Yaskawa INFORM job: OK_R2_O22-23(-90,180)OKKR.JBI

/JOB
//NAME OK_R2_O22-23(-90,180)OKKR
///FOLDERNAME X4
//POS
///NPOS 109,109,109,5,0,0
///TOOL 0
///POSTYPE PULSE
///PULSE
C00000=34467,8161,-3438,41001,63186,-12360
C00001=79400,-96450,-73119,47071,38510,-50576
C00002=120689,-37236,-43262,1430,36977,-65337
C00003=120661,8390,6118,1752,30038,-65509
C00004=121363,14227,14389,901,27936,-65072
C00005=121630,18134,20803,569,25994,-64899
C00006=122051,20456,22985,-52,25844,-64579
C00007=122335,22651,22887,209,31352,-64420
C00008=122335,23153,24532,213,30597,-64422
C00009=122573,22007,22272,-73,31399,-64269
C00010=118553,33336,34533,-32200,31167,-63632
C00011=118554,33797,35647,-32601,30785,-63423
C00012=118795,35881,37778,-33055,30674,-63177
C00013=119029,34698,36884,-33342,30719,-63021
C00014=119029,35470,39068,-34241,29924,-62556
C00015=119029,34698,36884,-33342,30719,-63021
C00016=122566,16275,19454,-818,25870,-64189
C00017=120682,5973,-10666,-26006,48512,-34380
C00018=120682,6077,-8041,-26626,47105,-33962
C00019=120965,19546,-3322,-22995,60520,-37308
C00020=120686,6056,-8291,-26571,47234,-33999
C00021=120521,4024,-8795,-26757,46523,-33864
C00022=122243,21545,4650,-37838,56763,-29509
C00023=115724,34900,14421,-35017,60862,-31707
C00024=115313,34877,14397,-34830,60697,-31836
C00025=122685,12952,-4874,-39297,55027,-28576
C00026=131885,-4518,-22891,-42927,60902,-26587
C00027=120689,-37236,-43262,1430,36977,-65337
C00028=79400,-96450,-73119,47071,38510,-50576
C00029=-8645,-72931,-67050,57733,95594,-74029
C00030=-3643,-76224,-106676,-19950,71810,-76872
C00031=-266,-73751,-67438,57600,90404,-72524
C00032=56065,-40103,-98025,15235,73272,-62938
C00033=80290,13979,-35130,8518,69424,-54762
C00034=81621,16186,-30024,7817,67316,-54480
C00035=82138,17140,-27919,7543,66474,-54366
C00036=82701,19213,-25983,7203,66302,-54190
C00037=82138,17140,-27919,7543,66474,-54366
C00038=82074,13923,-28800,7646,65378,-54460
C00039=82073,13446,-28104,7686,64710,-54504
C00040=82074,14344,-29367,7613,65938,-54423
C00041=80200,10192,-35655,8662,67827,-54907
C00042=80279,11679,-32768,3860,64531,-54120
C00043=80277,10318,-30958,3920,62722,-54182
C00044=80747,9882,-30077,3637,61936,-54046
C00045=80280,10347,-31011,3916,62769,-54180
C00046=79691,8209,-31623,4330,62077,-54408
C00047=80388,10283,-29809,3872,61992,-54168
C00048=75041,22104,-18783,7439,61626,-56057
C00049=80303,10454,-30913,3901,62763,-54172
C00050=80304,11819,-32719,3842,64572,-54110
C00051=56065,-40103,-98025,15235,73272,-62938
C00052=-3643,-76224,-106676,-19950,71810,-76872
C00053=-266,-73751,-67438,57600,90404,-72524
C00054=-266,-73751,-67438,57600,90404,-72524
C00055=-266,-73751,-67438,57600,90404,-72524
C00056=-266,-73751,-67438,57600,90404,-72524
C00057=-266,-73751,-67438,57600,90404,-72524
C00058=-266,-73751,-67438,57600,90404,-72524
C00059=-266,-73751,-67438,57600,90404,-72524
C00060=-266,-73751,-67438,57600,90404,-72524
C00061=-266,-73751,-67438,57600,90404,-72524
C00062=120677,-3480,-20614,18181,54095,39471
C00063=120311,11594,-4773,18885,52273,38972
C00064=120169,13967,1466,19666,49827,38417
C00065=119883,15460,2829,19877,49828,38285
C00066=119880,14569,2014,19868,49870,38293
C00067=119880,14692,3030,20029,49339,38180
C00068=119880,15002,5218,20385,48223,37938
C00069=119880,14692,3030,20029,49339,38180
C00070=121128,7117,-4698,18949,49860,38864
C00071=120984,8550,-10493,36755,60982,29079
C00072=120492,10444,-8592,38530,61785,27976
C00073=119910,12056,-7149,38807,61994,27785
C00074=120247,11117,-7991,38646,61874,27896
C00075=120247,11130,-6123,39024,60976,27528
C00076=120247,11117,-7991,38646,61874,27896
C00077=118757,6782,-7537,20091,51910,38210
C00078=120681,6612,-10378,25984,47448,35852
C00079=120681,6707,-7755,26629,46038,35426
C00080=120905,16102,-4997,22232,56693,38204
C00081=120839,4648,-8519,26766,45460,35327
C00082=120685,6692,-7997,26566,46163,35467
C00083=117786,13784,-6304,24852,56256,36873
C00084=124524,9883,-9298,30535,58908,31643
C00085=123624,18800,-2226,35492,64552,29693
C00086=120681,6624,-6675,42630,54896,24176
C00087=115739,6767,-11022,43739,59328,23743
C00088=-266,-73751,-67438,57600,90404,-72524
C00089=-266,-73751,-67438,57600,90404,-72524
C00090=73074,14271,-65905,40005,100084,34925
C00091=80386,15191,-35510,35923,83035,31364
C00092=81077,18148,-29671,35761,81084,30977
C00093=80079,11495,-28631,39585,73800,28709
C00094=80398,13741,-26603,39455,73592,28760
C00095=80079,11495,-28631,39585,73800,28709
C00096=81415,17339,-25976,35859,78754,30337
C00097=81415,16938,-25408,35919,78297,30186
C00098=80477,16259,-27610,36210,79478,30223
C00099=80390,10982,-30842,41019,80930,29700
C00100=75774,13099,-22819,50986,80482,25907
C00101=80082,8484,-31856,41199,80558,29427
C00102=80393,11011,-30897,41013,80966,29715
C00103=75635,11609,-22454,52738,79251,24739
C00104=81623,6978,-27251,49926,76964,26328
C00105=82021,7248,-27571,49491,77489,26755
C00106=80364,10836,-30874,41034,80899,29677
C00107=80366,12212,-32666,40889,82284,30221
C00108=73074,14271,-65905,40005,100084,34925
BC00000=125683,503280,458302
BC00001=125909,496171,117576
BC00002=159989,496171,117576
BC00003=159989,496171,117576
BC00004=159989,496171,117576
BC00005=159989,496171,117576
BC00006=159989,496171,117576
BC00007=159989,496171,117576
BC00008=159989,496171,117576
BC00009=159989,496171,117576
BC00010=159989,496171,117576
BC00011=159989,496171,117576
BC00012=159989,496171,117576
BC00013=159989,496171,117576
BC00014=159989,496171,117576
BC00015=159989,496171,117576
BC00016=159989,496171,117576
BC00017=109858,489893,17
BC00018=109452,483826,17
BC00019=109349,482285,17
BC00020=109289,481399,17
BC00021=109289,481399,17
BC00022=161912,473661,17
BC00023=161912,473661,17
BC00024=161912,473661,17
BC00025=161912,473661,17
BC00026=161912,473661,17
BC00027=159989,496171,117576
BC00028=125909,496171,117576
BC00029=97158,510235,426323
BC00030=199448,515539,1075137
BC00031=97158,523229,1005604
BC00032=48431,468399,1061681
BC00033=36737,455240,1075139
BC00034=36737,455240,1075139
BC00035=36737,455240,1075139
BC00036=36737,455240,1075139
BC00037=36737,455240,1075139
BC00038=36737,455240,1075139
BC00039=36737,455240,1075139
BC00040=36737,455240,1075139
BC00041=36737,455240,1075139
BC00042=22763,453119,1075139
BC00043=22467,447673,1075139
BC00044=22349,445495,1075139
BC00045=22349,445495,1075139
BC00046=22349,445495,1075139
BC00047=64148,438226,1075139
BC00048=64148,438226,1075139
BC00049=64267,440404,1075139
BC00050=64562,445850,1075139
BC00051=48431,468399,1061681
BC00052=199448,515539,1075137
BC00053=97158,523229,1005604
BC00054=97158,523229,922174
BC00055=97158,523229,922174
BC00056=97158,523229,918568
BC00057=97158,523229,720053
BC00058=97158,523229,697581
BC00059=97158,523229,697581
BC00060=97158,523229,426323
BC00061=97158,523229,426323
BC00062=311340,483475,69287
BC00063=311340,483475,69287
BC00064=311340,483475,69287
BC00065=311340,483475,69287
BC00066=311340,483475,69287
BC00067=311340,483475,69287
BC00068=311340,483475,69287
BC00069=311340,483475,69287
BC00070=311340,483475,69287
BC00071=275671,458791,6419
BC00072=272431,456549,709
BC00073=272431,456549,709
BC00074=272431,456549,709
BC00075=272431,456549,709
BC00076=272431,456549,709
BC00077=311340,483475,69287
BC00078=328863,490903,17
BC00079=329302,484845,17
BC00080=329445,482870,17
BC00081=329478,482421,17
BC00082=329478,482421,17
BC00083=268709,471953,17
BC00084=272116,455909,17
BC00085=272116,455909,17
BC00086=272765,458336,17
BC00087=274387,464402,17
BC00088=97158,523229,426323
BC00089=97158,523229,1033177
BC00090=194066,506419,1075139
BC00091=194066,454256,1075139
BC00092=194066,454256,1075139
BC00093=194066,454256,1075139
BC00094=194066,454256,1075139
BC00095=194066,454256,1075139
BC00096=194066,454256,1075139
BC00097=194066,454256,1075139
BC00098=194066,454256,1075139
BC00099=207734,447131,1075139
BC00100=207866,444951,1075138
BC00101=207866,444951,1075139
BC00102=207866,444951,1075139
BC00103=170759,438554,1075139
BC00104=170759,438554,1075139
BC00105=170759,438554,1075139
BC00106=165921,439933,1075139
BC00107=165591,445383,1075139
BC00108=194066,506419,1075139
EC00000=798152,-1296784
EC00001=798156,-1296783
EC00002=798156,-1296783
EC00003=798156,-1296783
EC00004=798156,-1296783
EC00005=798156,-1296783
EC00006=798156,-1296783
EC00007=798156,-1296783
EC00008=798156,-1296783
EC00009=798156,-1296783
EC00010=798156,-1296783
EC00011=798156,-1296783
EC00012=798156,-1296783
EC00013=798156,-1296783
EC00014=798156,-1296783
EC00015=798156,-1296783
EC00016=798156,-1296783
EC00017=798156,-1296783
EC00018=798156,-1296783
EC00019=798156,-1296783
EC00020=798156,-1296783
EC00021=798156,-1296783
EC00022=798156,-1296783
EC00023=798156,-1296783
EC00024=798156,-1296783
EC00025=798156,-1296783
EC00026=798156,-1296783
EC00027=798156,-1296783
EC00028=798156,-1296783
EC00029=798156,-1296783
EC00030=798156,-1296783
EC00031=798156,-1296783
EC00032=798156,-1296783
EC00033=798156,-1296783
EC00034=798156,-1296783
EC00035=798156,-1296783
EC00036=798156,-1296783
EC00037=798156,-1296783
EC00038=798156,-1296783
EC00039=798156,-1296783
EC00040=798156,-1296783
EC00041=798156,-1296783
EC00042=798156,-1296783
EC00043=798156,-1296783
EC00044=798156,-1296783
EC00045=798156,-1296783
EC00046=798156,-1296783
EC00047=798156,-1296783
EC00048=798156,-1296783
EC00049=798156,-1296783
EC00050=798156,-1296783
EC00051=798156,-1296783
EC00052=798156,-1296783
EC00053=798156,-1296783
EC00054=861922,-1136491
EC00055=880722,-998760
EC00056=879279,-887535
EC00057=885682,-601799
EC00058=877307,-527453
EC00059=877307,-423086
EC00060=798156,-183832
EC00061=798156,-183832
EC00062=798156,-183832
EC00063=798156,-183832
EC00064=798156,-183832
EC00065=798156,-183832
EC00066=798156,-183832
EC00067=798156,-183832
EC00068=798156,-183832
EC00069=798156,-183832
EC00070=798156,-183832
EC00071=798156,-183832
EC00072=798156,-183832
EC00073=798156,-183832
EC00074=798156,-183832
EC00075=798156,-183832
EC00076=798156,-183832
EC00077=798156,-183832
EC00078=798156,-183832
EC00079=798156,-183832
EC00080=798156,-183832
EC00081=798156,-183832
EC00082=798156,-183832
EC00083=798156,-183832
EC00084=798156,-183832
EC00085=798156,-183832
EC00086=798156,-183832
EC00087=798156,-183832
EC00088=798156,-183832
EC00089=798156,-183832
EC00090=798156,-183832
EC00091=798156,-183832
EC00092=798156,-183832
EC00093=798156,-183832
EC00094=798156,-183832
EC00095=798156,-183832
EC00096=798156,-183832
EC00097=798156,-183832
EC00098=798156,-183832
EC00099=798156,-183832
EC00100=798154,-183832
EC00101=798156,-183832
EC00102=798156,-183832
EC00103=798156,-183832
EC00104=798156,-183832
EC00105=798156,-183832
EC00106=798156,-183832
EC00107=798156,-183832
EC00108=798156,-183832
///POSTYPE BASE
///RECTAN
///RCONF 0,0,0,0,1,0,0,0,0,0,0,0,0,0,0,0,0,0,0,0,0,0,0,0
P00006=2.006,1.622,-0.565,0.0000,0.0000,0.0000
P00021=0.073,2.058,-0.109,0.0000,0.0000,0.0000
P00022=2.006,1.622,-0.565,0.0000,0.0000,0.0000
///RCONF 0,0,0,0,0,0,0,0,0,0,0,0,0,0,0,0,0,0,0,0,0,0,0,0
P00023=-2.957,-4.083,2.762,0.0000,0.0000,0.0000
P00024=-1.466,-0.226,-0.419,0.0000,0.0000,0.0000
//INST
///DATE 2024/11/25 16:22
///ATTR SC,RW
///GROUP1 RB1,BS1
///GROUP2 ST1
NOP
'OK_r2_O22-23(-90,180)
MOVJ C00000 BC00000 VJ=50.00  +MOVJ EC00000 VJ=50.00
MOVJ C00001 BC00001 VJ=100.00  +MOVJ EC00001 VJ=100.00
MOVJ C00002 BC00002 VJ=100.00  +MOVJ EC00002 VJ=100.00
'Path S1012
SFTOF3D
MOVJ C00003 BC00003 VJ=100.00  +MOVJ EC00003 VJ=100.00
MOVL C00004 BC00004 V=400.0  +MOVJ EC00004 VJ=100.00
SMOVL C00005 BC00005 V=133.3  +MOVJ EC00005
SREFP 3 C00006 BC00006  +REFP EC00006
CALL JOB:SEARCH-R1-S13D
SET P023 P006
SFTON3D P023
SMOVL C00007 BC00007 V=133.3  +MOVJ EC00007
SREFP 3 C00008 BC00008  +REFP EC00008
CALL JOB:SEARCH-R1-S13D
SET P023 P006
SFTON3D P023
SMOVL C00009 BC00009 V=166.7  +MOVJ EC00009
SFTOF3D
SMOVL C00010 BC00010 V=416.7  +MOVJ EC00010
SMOVL C00011 BC00011 V=166.7  +MOVJ EC00011
SREFP 3 C00012 BC00012  +REFP EC00012
CALL JOB:SEARCH-R1-S13D
SET P024 P006
SFTON3D P024
SMOVL C00013 BC00013 V=133.3  +MOVJ EC00013
SREFP 3 C00014 BC00014  +REFP EC00014
CALL JOB:SEARCH-R1-S13D
SET P024 P006
SFTON3D P024
SMOVL C00015 BC00015 V=166.7  +MOVJ EC00015
SFTOF3D
MOVL C00016 BC00016 V=400.0  +MOVJ EC00016 VJ=100.00
'Path W1013
SFTOF3D
SFTON3D P023
MOVJ C00017 BC00017 VJ=100.00  +MOVJ EC00017 VJ=100.00
SMOVL C00018 BC00018 V=400.0  +MOVJ EC00018
SMOVL C00019 BC00019 V=133.3 PL=0  +MOVJ EC00019
SREFP 1 C00020 BC00020  +REFP EC00020
SREFP 2 C00021 BC00021  +REFP EC00021
MACRO1 MJ#(0) ARGF6
ARCON
SFTON3D P024
SMOVL C00022 BC00022 V=7.5  +MOVJ EC00022
SMOVL C00023 BC00023 V=7.5  +MOVJ EC00023
ARCON
SMOVL C00024 BC00024 V=7.5  +MOVJ EC00024
ARCOF
SMOVL C00025 BC00025 V=400.0  +MOVJ EC00025
SMOVL C00026 BC00026 V=1000.0  +MOVJ EC00026
SFTOF3D
MOVJ C00027 BC00027 VJ=100.00  +MOVJ EC00027 VJ=100.00
MOVJ C00028 BC00028 VJ=100.00  +MOVJ EC00028 VJ=100.00
MOVJ C00029 BC00029 VJ=100.00  +MOVJ EC00029 VJ=100.00
'R-L Trip
MOVJ C00030 BC00030 VJ=100.00  +MOVJ EC00030 VJ=100.00
CALL JOB:CLEAN-R1_KM_NEW
MOVJ C00031 BC00031 VJ=100.00  +MOVJ EC00031 VJ=100.00
MOVJ C00032 BC00032 VJ=100.00  +MOVJ EC00032 VJ=100.00
'Path S1396
SFTOF3D
MOVJ C00033 BC00033 VJ=100.00  +MOVJ EC00033 VJ=100.00
MOVL C00034 BC00034 V=333.3  +MOVJ EC00034 VJ=100.00
SMOVL C00035 BC00035 V=166.7  +MOVJ EC00035
SREFP 3 C00036 BC00036  +REFP EC00036
CALL JOB:SEARCH-R1-S13D
SET P024 P006
SFTON3D P024
SMOVL C00037 BC00037 V=166.7  +MOVJ EC00037
SMOVL C00038 BC00038 V=166.7  +MOVJ EC00038
SREFP 3 C00039 BC00039  +REFP EC00039
CALL JOB:SEARCH-R1-S13D
SET P024 P006
SFTON3D P024
SMOVL C00040 BC00040 V=166.7  +MOVJ EC00040
MOVL C00041 BC00041 V=1000.0  +MOVJ EC00041 VJ=100.00
'Path W1397
SFTOF3D
SFTON3D P024
MOVJ C00042 BC00042 VJ=100.00  +MOVJ EC00042 VJ=100.00
SMOVL C00043 BC00043 V=400.0  +MOVJ EC00043
SMOVL C00044 BC00044 V=166.7 PL=0  +MOVJ EC00044
SREFP 1 C00045 BC00045  +REFP EC00045
SREFP 2 C00046 BC00046  +REFP EC00046
MACRO1 MJ#(0) ARGF6
ARCON
SMOVL C00047 BC00047 V=8.3  +MOVJ EC00047
SMOVL C00048 BC00048 V=8.3  +MOVJ EC00048
ARCOF
SMOVL C00049 BC00049 V=400.0  +MOVJ EC00049
SMOVL C00050 BC00050 V=1000.0  +MOVJ EC00050
SFTOF3D
MOVJ C00051 BC00051 VJ=100.00  +MOVJ EC00051 VJ=100.00
MOVJ C00052 BC00052 VJ=100.00  +MOVJ EC00052 VJ=100.00
CALL JOB:CLEAN-R1_KM_NEW
MOVJ C00053 BC00053 VJ=100.00  +MOVJ EC00053 VJ=100.00
MOVJ C00054 BC00054 VJ=100.00  +MOVJ EC00054 VJ=100.00
MOVJ C00055 BC00055 VJ=100.00  +MOVJ EC00055 VJ=100.00
MOVJ C00056 BC00056 VJ=100.00  +MOVJ EC00056 VJ=100.00
MOVJ C00057 BC00057 VJ=100.00  +MOVJ EC00057 VJ=100.00
MOVJ C00058 BC00058 VJ=100.00  +MOVJ EC00058 VJ=100.00
MOVJ C00059 BC00059 VJ=100.00  +MOVJ EC00059 VJ=100.00
MOVJ C00060 BC00060 VJ=100.00  +MOVJ EC00060 VJ=100.00
MOVJ C00061 BC00061 VJ=100.00  +MOVJ EC00061 VJ=100.00
'Path S1392
SFTOF3D
MOVJ C00062 BC00062 VJ=100.00  +MOVJ EC00062 VJ=100.00
MOVL C00063 BC00063 V=166.7  +MOVJ EC00063 VJ=100.00
SMOVL C00064 BC00064 V=166.7  +MOVJ EC00064
SREFP 3 C00065 BC00065  +REFP EC00065
CALL JOB:SEARCH-R1-S13D
SET P021 P006
SFTON3D P021
SMOVL C00066 BC00066 V=166.7  +MOVJ EC00066
SMOVL C00067 BC00067 V=166.7  +MOVJ EC00067
SREFP 3 C00068 BC00068  +REFP EC00068
CALL JOB:SEARCH-R1-S13D
SET P021 P006
SFTON3D P021
SMOVL C00069 BC00069 V=166.7  +MOVJ EC00069
SFTOF3D
MOVL C00070 BC00070 V=400.0  +MOVJ EC00070 VJ=100.00
SMOVL C00071 BC00071 V=666.7  +MOVJ EC00071
SMOVL C00072 BC00072 V=166.7  +MOVJ EC00072
SREFP 3 C00073 BC00073  +REFP EC00073
CALL JOB:SEARCH-R1-S13D
SET P022 P006
SFTON3D P022
SMOVL C00074 BC00074 V=166.7  +MOVJ EC00074
SREFP 3 C00075 BC00075  +REFP EC00075
CALL JOB:SEARCH-R1-S13D
SET P022 P006
SFTON3D P022
SMOVL C00076 BC00076 V=166.7  +MOVJ EC00076
MOVL C00077 BC00077 V=1000.0  +MOVJ EC00077 VJ=100.00
'Path W1393
SFTOF3D
SFTON3D P021
MOVJ C00078 BC00078 VJ=100.00  +MOVJ EC00078 VJ=100.00
SMOVL C00079 BC00079 V=400.0  +MOVJ EC00079
SMOVL C00080 BC00080 V=166.7 PL=0  +MOVJ EC00080
SREFP 1 C00081 BC00081  +REFP EC00081
SREFP 2 C00082 BC00082  +REFP EC00082
MACRO1 MJ#(0) ARGF6
ARCON
SFTON3D P022
SMOVL C00083 BC00083 V=7.5  +MOVJ EC00083
SMOVL C00084 BC00084 V=7.5  +MOVJ EC00084
SMOVL C00085 BC00085 V=7.5  +MOVJ EC00085
ARCOF
SFTOF3D
SMOVL C00086 BC00086 V=400.0  +MOVJ EC00086
SMOVL C00087 BC00087 V=1000.0  +MOVJ EC00087
SFTOF3D
'L-R Trip
MOVJ C00088 BC00088 VJ=100.00  +MOVJ EC00088 VJ=100.00
CALL JOB:CLEAN-R1_KM_NEW
MOVJ C00089 BC00089 VJ=100.00  +MOVJ EC00089 VJ=100.00
MOVJ C00090 BC00090 VJ=100.00  +MOVJ EC00090 VJ=100.00
'Path S1394
SFTOF3D
MOVJ C00091 BC00091 VJ=100.00  +MOVJ EC00091 VJ=100.00
MOVL C00092 BC00092 V=400.0  +MOVJ EC00092 VJ=100.00
SMOVL C00093 BC00093 V=166.7  +MOVJ EC00093
SREFP 3 C00094 BC00094  +REFP EC00094
CALL JOB:SEARCH-R1-S13D
SET P022 P006
SFTON3D P022
SMOVL C00095 BC00095 V=166.7  +MOVJ EC00095
SMOVL C00096 BC00096 V=166.7  +MOVJ EC00096
SREFP 3 C00097 BC00097  +REFP EC00097
CALL JOB:SEARCH-R1-S13D
SET P022 P006
SFTON3D P022
SMOVL C00098 BC00098 V=166.7  +MOVJ EC00098
'Path W1395
SFTOF3D
SFTON3D P022
SMOVL C00099 BC00099 V=400.0  +MOVJ EC00099
SMOVL C00100 BC00100 V=166.7 PL=0  +MOVJ EC00100
SREFP 1 C00101 BC00101  +REFP EC00101
SREFP 2 C00102 BC00102  +REFP EC00102
MACRO1 MJ#(0) ARGF6
ARCON
SMOVL C00103 BC00103 V=7.5  +MOVJ EC00103
SMOVL C00104 BC00104 V=7.5  +MOVJ EC00104
SMOVL C00105 BC00105 V=7.5  +MOVJ EC00105
ARCOF
SMOVL C00106 BC00106 V=400.0  +MOVJ EC00106
SMOVL C00107 BC00107 V=1000.0  +MOVJ EC00107
SFTOF3D
MOVJ C00108 BC00108 VJ=100.00  +MOVJ EC00108 VJ=100.00
END
